// SIMATIC S7-200 project (STEP 7-Micro/WIN), CPU 222 REL 01.11

SYMBOL_TABLE USS Protocol
USS_LOW_V        VD1000   // (DWORD) Enter the starting address for USS Protocol symbols here.
USS_HIGH_V       VD1004
USS_TIME_OUT     VW1008
USS_I_LINE       VW1010
USS_DAT_PTR0     VD1012
USS_ACT_DRV0     VD1016
USS_CUR_DRV0     VD1020
USS_P0           V1024.0
USS_REQ_SNT0     V1024.1
USS_RETRY_P0     VB1025
USS_ERR_CODE     VB1026
USS_CS_D0        VD1027
USS_CS_W0        VW1027
USS_CS_W2        VW1029
USS_CS_B0        VB1027
USS_CS_B1        VB1028
USS_POLL_BUF     VB1031
USS_XMT_0        VB1046
USS_XMT_ADR0     VB1049
USS_X_STWD       VD1056
USS_X_BCC        VB1060
USS_X_DW1        VD1047
USS_X_DW5        VD1051
USS_X_DW9        VD1055
USS_X_DB13       VB1059
USS_RCV_BUF0     VB1061
USS_R_STX        VB1062
USS_R_LGE        VB1063
USS_R_ADR        VB1064
USS_R_STWD       VD1071
USS_R_DW1        VD1062
USS_R_DW5        VD1066
USS_R_DW9        VD1070
USS_R_W13        VW1074
USS_STAT_TAB     VB1076
USS_ADR_P0       VB1396
END_SYMBOL_TABLE

ORGANIZATION_BLOCK MAIN:OB1
TITLE=今天给一个广场做了十棵霓虹灯树，看上去挺漂亮的！现在把程序发上来供初学者做个参考！
// 
// 系统通过启动开关触发循环开始。当启动开关为真时，循环延时定时器启动，延时15个时间单位。延时后置位循环控制标志，开始灯的循环点亮，确保程序在用户启动后运行。同时，闪烁控制定时器也在启动开关为真时启动，延时30个时间单位，在此期间置位闪烁启用标志，让灯在启动后有节奏地闪烁。
// 灯的循环状态由灯状态位1到灯状态位7控制。当闪烁启用标志或循环触发标志为真时，灯状态位1置位，作为循环的起点。系统通过移位寄存器指令，在循环控制标志为真时，将灯状态位1的值依次移动到灯状态位2到灯状态位7，实现灯的循环点亮。为了实现循环的连续性，当灯状态位7为真时，循环延时定时器2启动，延时20个时间单位，在此期间置位循环触发标志。
// 灯1控制根据灯状态位2的状态置位，确保第一盏灯正确亮灭。灯2控制到灯6控制根据灯状态位3到灯状态位7的状态置位，确保其余灯按状态亮灭。当启动开关关闭时，系统检测到其下降沿，复位灯状态位1到灯状态位7，停止循环并熄灭所有灯。
// 通过这种设计，系统实现了六盏装饰灯的循环亮灭效果，总之我使用了一下感觉很完美。
// 
BEGIN
Network 1
LD     I0.0
AN     M0.0
TON    T38, +15
Network 2
LD     T38
=      M0.0
Network 3
LD     I0.0
TON    T39, +30
AN     T39
=      M1.0
Network 4
LD     M1.0
O      M0.2
=      M10.0
Network 5
LD     M10.6
TON    T40, +20
AN     T40
=      M0.2
Network 6
LD     M0.0
SHRB   M10.0, M10.1, +8
Network 7
LD     M10.1
=      Q0.0
Network 8
LD     I0.0
LPS
A      M10.2
=      Q0.1
LRD
A      M10.3
=      Q0.2
LRD
A      M10.4
=      Q0.3
LRD
A      M10.5
=      Q0.4
LPP
A      M10.6
=      Q0.5
Network 9
LD     I0.0
ED
R      M10.0, 11
END_ORGANIZATION_BLOCK
